// Mitsubishi GX Works2 project: 230930-001- de hoje   PLC: Q03UDV

// task Task_01 (event TRUE, interval 0, priority 31): POU_01

PROGRAM POU_01
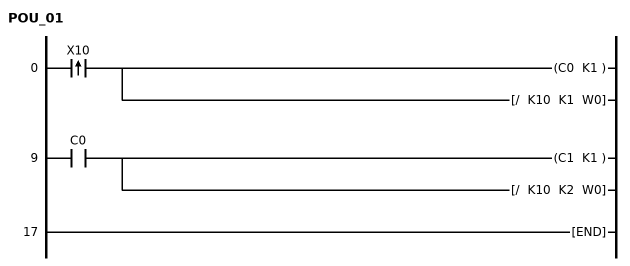
0     LDP     X10
      OUT     C0 K1
      /       K10 K1 W0
9     LD      C0
      OUT     C1 K1
      /       K10 K2 W0
17    END
END_PROGRAM
